// TIA Portal V16 program export: 1 tag tables, 0 data types, 20 data blocks, 10 code blocks (in call order from the OBs), 24 instance data blocks

VAR_GLOBAL   // PLC tag table "Default tag table"
   Iniciar_Manual AT %I0.0 : Bool;
   Detener_Manual AT %I0.1 : Bool;
   Raw_Temperatura AT %IW64 : Int;
   Raw_Humedad AT %IW66 : Int;
   Deshidratador AT %Q0.0 : Bool;
   Actuador AT %Q0.1 : Bool;
   Ventilador AT %Q0.2 : Bool;
   Resistencias AT %Q0.3 : Bool;
   Sensor_Modbus AT %Q0.4 : Bool;
   Sensor_HT AT %Q0.5 : Bool;
   System_Byte AT %MB1 : Byte;
   FirstScan AT %M1.0 : Bool;
   DiagStatusUpdate AT %M1.1 : Bool;
   AlwaysTRUE AT %M1.2 : Bool;
   AlwaysFALSE AT %M1.3 : Bool;
   Clock_Byte AT %MB0 : Byte;
   Clock_10Hz AT %M0.0 : Bool;
   Clock_5Hz AT %M0.1 : Bool;
   "Clock_2.5Hz" AT %M0.2 : Bool;
   Clock_2Hz AT %M0.3 : Bool;
   "Clock_1.25Hz" AT %M0.4 : Bool;
   Clock_1Hz AT %M0.5 : Bool;
   "Clock_0.625Hz" AT %M0.6 : Bool;
   "Clock_0.5Hz" AT %M0.7 : Bool;
   Control_Byte AT %MB2 : Byte;
   Detener AT %M2.0 : Bool;
   Iniciar AT %M2.1 : Bool;
   Pausar AT %M2.2 : Bool;
   Activar_Deshidratador AT %M2.3 : Bool;
   Limite_Matte AT %M2.6 : Bool;
   Sensor_Modbus_Manual AT %M2.4 : Bool;
   Set_Point_Deshidratador AT %MD4 : Real;
   Set_Point_Humedad AT %MD8 : Real;
   Iniciar_Pulse AT %M30.0 : Bool;
   Detener_Pulse AT %M30.1 : Bool;
   Guardar_Datos AT %M30.2 : Bool;
   Data_Log_Write_Error AT %M30.3 : Bool;
   Data_Log_Write_Busy AT %M30.4 : Bool;
   Data_Log_Write_Done AT %M30.5 : Bool;
   Data_Log_Write_Status AT %MW34 : Word;
   "Clock_0.016Hz" AT %M30.6 : Bool;
   Ret_Val AT %MW36 : Int;
   Sensor_HT_Manual AT %M2.5 : Bool;
   Actuador_Manual AT %M2.7 : Bool;
   Activar_Actuador AT %M3.0 : Bool;
   Tag_1 AT %M31.1 : Bool;
   Habilitar_Matte AT %M3.1 : Bool;
   Set_Point_Limite AT %MD12 : Real;
   Humedad_Material_D11 AT %MD38 : Real;
   Humedad_Material_D13 AT %MD42 : Real;
   Humedad_Material_D16 AT %MD46 : Real;
   Temp_D13 AT %MD54 : Real;
   Temp_Matte AT %MD58 : Real;
   Hum_Matte AT %MD62 : Real;
   Temp_D11 AT %MD50 : Real;
   Temp_Matte_Aux AT %MD66 : Real;
   Clock_Matte_Manual AT %M31.2 : Bool;
   Humedad_Material_D11_Ajuste AT %MD70 : Real;
   Humedad_Material_D13_Ajuste AT %MD74 : Real;
   Humedad_Material_D16_Ajuste AT %MD78 : Real;
   Hum_Matte_Aux AT %MD82 : Real;
   Random_Real_Seconds AT %MD86 : Real;
   Random_Status AT %MW90 : Int;
   Random_Sub_Status AT %MW92 : Int;
   Random_Error AT %M3.2 : Bool;
   Clock_Pulse AT %M3.3 : Bool;
   Randon_Dint_Seconds AT %MD94 : DInt;
   Tiempo_Histeresis_D1 AT %MD98 : Time;
   Set_Point_Deshidratador1_Inicial AT %MD102 : Real;
   Set_Point_Deshidratador1_Intermedia AT %MD106 : Real;
   Set_Point_Deshidratador1_Final AT %MD110 : Real;
   Set_Point_Humedad_D1_Inicial AT %MD114 : Real;
   Set_Point_Humedad_D1_Intermedia AT %MD118 : Real;
   Set_Point_Humedad_D1_Final AT %MD122 : Real;
   Detener_Desde_Modo_Preset AT %M31.3 : Bool;
END_VAR
VAR_GLOBAL CONSTANT   // user constants
   Set_Point_Temp_Default : Real := 55.0;
   Set_Pont_Hum_Default : Real := 5.0;
   Set_Point_Lim_Default : Real := -16.0;
   Aux_Hum_D1 : Real := 10.0;
   Aux_Hum_D4 : Real := 25.0;
   Aux_Hum_D8 : Real := 25.0;
END_VAR

DATA_BLOCK "Alarmas"   // DB44
{ S7_Optimized_Access := 'FALSE' }
VERSION : 0.1
   VAR
      Alarma_Fin_Operacion : Bool;
      Alarma_Fallo_Deh : Bool;
   END_VAR
BEGIN
END_DATA_BLOCK

DATA_BLOCK "CREAR_DB"   // DB7
{ S7_Optimized_Access := 'TRUE' }
VERSION : 0.1
   VAR
      records : UDInt := 17280;
      "name" : String := 'logging';
      id : DWord := 1;
      headers : String := 'HumD11,HumD13,HumD16,TempD11,TempD13,HumMatte,TempMatte';
      data : Struct
         humD11 : Real;
         humD13 : Real;
         humD16 : Real;
         tempD11 : Real;
         tempD13 : Real;
         humMatte : Real;
         tempMatte : Real;
      END_STRUCT;
      done : Bool;
      busy : Bool := true;
      error : Bool;
      status : Word;
   END_VAR
BEGIN
END_DATA_BLOCK

DATA_BLOCK "Calibracion_Sensores"   // DB31
{ S7_Optimized_Access := 'TRUE' }
VERSION : 0.1
   VAR
      Ajuste_D11 : Real := 1.0;
      Ajuste_D13 : Real := 1.0;
      Ajuste_D16 : Real := 1.0;
      Ajuste_T1 : Real := 1.0;
   END_VAR
BEGIN
END_DATA_BLOCK

DATA_BLOCK "Control_Log_DB"   // DB33
{ S7_Optimized_Access := 'FALSE' }
VERSION : 0.1
   VAR
      Iniciar_Log : Bool;
      Almacenar_Logs : Bool;
      Teminar_Log : Bool;
   END_VAR
BEGIN
END_DATA_BLOCK

DATA_BLOCK "DATOS_MODSEC"   // DB13
{ S7_Optimized_Access := 'TRUE' }
VERSION : 0.1
   VAR
      SimuHR : Int;
   END_VAR
   VAR RETAIN
      "Paso Control HR" : Time := T#5000ms;
      "Paso Grafica" : Time := T#10ms;
      "CRECIMIENTO HR" : Real := 80.0;
      TempMinHR : Real := 22.0;
   END_VAR
   VAR
      TempInf : Real := 0.0;
      TempSup : Real := 100.0;
      TempFilt : Real;
      TempFiltJP : Real;
      HRAux : Real;
      HRAuxJP : Real;
      HRFilt : Real;
      HRSim : Int;
      TempSim : Int;
      ProporcionHumedad : Real := 0.9;
      TempFiltCuar : Real;
      HRFiltCuar : Real;
      HRAuxCuar : Real;
   END_VAR
BEGIN
END_DATA_BLOCK

DATA_BLOCK "DATOS_VARIABLES"   // DB8
{ S7_Optimized_Access := 'FALSE' }
VERSION : 0.1
   VAR
      humD11 : Real;
      humD13 : Real;
      humD16 : Real;
      tempD11 : Real;
      tempD13 : Real;
      humMatte : Real;
      tempMatte : Real;
   END_VAR
BEGIN
END_DATA_BLOCK

DATA_BLOCK "MB_CONFIG"   // DB9
{ S7_Optimized_Access := 'FALSE' }
VERSION : 0.1
   VAR
      Again : Bool;
      Req : Bool;
      Mb_Addr : UInt := 1;
      Mode : USInt := 0;
      Data_Addr : UDInt := 40001;
      Data_Len : UInt := 5;
      Done : Bool;
      Busy : Bool;
      Error : Bool;
      Status : Word;
      Error_Status : Word;
      "Step" : Int := 1;
   END_VAR
BEGIN
END_DATA_BLOCK

DATA_BLOCK "MB_DATA_BUFFER"   // DB10
{ S7_Optimized_Access := 'FALSE' }
VERSION : 0.1
   VAR
      REGISTERS : Array[0..4] of UInt;
   END_VAR
BEGIN
END_DATA_BLOCK

DATA_BLOCK "MB_LOAD"   // DB11
{ S7_Optimized_Access := 'FALSE' }
VERSION : 0.1
   VAR
      Baud : UDInt := 9600;
      Parity : UDInt;
      Done : Bool;
      Error : Bool;
      Status : Word;
      Done_Stored : Bool;
      Error_Stored : Bool;
      Status_Error : Word;
   END_VAR
BEGIN
END_DATA_BLOCK

DATA_BLOCK "Modos_Operacion"   // DB32
{ S7_Optimized_Access := 'TRUE' }
VERSION : 0.1
   VAR
      Modo_Preset_D1 : Bool;
      Momento_Actual_D1 : Int;
   END_VAR
BEGIN
END_DATA_BLOCK

DATA_BLOCK "DB 333"   // DB333
{ S7_Optimized_Access := 'FALSE' }
AUTHOR : AWP_S7P
FAMILY : WEB
VERSION : 1.0
   VAR
      magic : DWord := DW#16#41575043;
      consistency_tag : DWord := DW#16#24B8E9AC;
      db_version : Word := W#16#0001;
      length : UInt := 4326;
      pagetab_of : UInt := 92;
      pagetab_count : UInt := 36;
      excludetab_of : UInt := 452;
      excludetab_count : UInt := 4;
      fragmentlist_of : UInt := 460;
      fragmentlist_count : UInt := 55;
      fragmenttab_of : UInt := 576;
      fragmenttab_count : UInt := 45;
      datatab_of : UInt := 1206;
      datatab_count : UInt := 30;
      usenametab_of : UInt := 1326;
      usenametab_count : UInt := 0;
      enumreftab_of : UInt := 1326;
      enumreftab_count : UInt := 0;
      enumtab_of : UInt := 1326;
      enumtab_count : UInt := 0;
      textlist_of : UInt := 1326;
      textlist_count : UInt := 3000;
      language_frag_tab_of : UInt := 570;
      language_frag_tab_count : UInt := 6;
      application_name : UInt := 1;
      application_url : UInt := 17;
      application_desc : UInt := 34;
      enum_defs_fragment_start : UInt := 0;
      enum_defs_fragment_count : UInt := 0;
      commandstate : Struct
         last_error : Int := 0;
         debug_mode : Int := 0;
         init : Bool := True;
         deactivate : Bool := False;
         initializing : Bool := False;
         error : Bool := False;
         deactivating : Bool := False;
         deactivated : Bool := False;
         initialized : Bool := False;
         reserved1 : Bool := False;
         reserved2 : Byte := B#16#00;
      END_STRUCT;
      requesttab : Array[1..4] of Struct
         page_index : UInt;
         fragment_index : UInt;
         continue : Bool;
         "repeat" : Bool;
         abort : Bool;
         finish : Bool;
         idle : Bool;
         waiting : Bool;
         sending : Bool;
         aborting : Bool;
         reserved3 : Byte;
      END_STRUCT;
      pagetab : Array[1..36] of Struct
         index : UInt;
         url : UInt;
         mime_type : UInt;
         fragment_start : UInt;
         fragment_num : UInt;
      END_STRUCT;
      excludetab : Array[1..4] of UInt;
      fragmentlist : Array[1..55] of UInt;
      language_frag_tab : Struct
         max_language : UInt := 0;
         fragment_count : UInt := 0;
         nolang_offset : UInt := 0;
      END_STRUCT;
      fragmenttab : Array[1..45] of Struct
         fragment_name : UInt;
         fragment_type : Byte;
         fragment_version : Byte;
         content_db : UInt;
         content_of : UInt;
         content_length : UInt;
         data_start : UInt;
         data_num : UInt;
      END_STRUCT;
      datatab : Array[1..30] of Struct
         variable_name : UInt;
         direction : Int;
      END_STRUCT;
      textlist : Array[1..3000] of Byte := 5365727669646F725175616E74756D0076696577735C6C6F67696E2E68746D6C005365727669646F725175616E74756D00494F4431487973745374617475732E68746D6C00746578742F68746D6C00494F44314D6F64652E68746D6C00746578742F68746D6C00494F44315374617475732E68746D6C00746578742F68746D6C00494F4465685374617475732E68746D6C00746578742F68746D6C00494F48756D4431312E68746D6C00746578742F68746D6C00494F48756D443146696E616C5374617475732E68746D6C00746578742F68746D6C00494F48756D4431496E69745374617475732E68746D6C00746578742F68746D6C00494F48756D44314D69645374617475732E68746D6C00746578742F68746D6C00494F48756D44315374617475732E68746D6C00746578742F68746D6C00494F53746172744465682E68746D6C00746578742F68746D6C00494F53746F704465682E68746D6C00746578742F68746D6C00494F54656D7044312E68746D6C00746578742F68746D6C00494F54656D70443146696E616C5374617475732E68746D6C00746578742F68746D6C00494F54656D704431496E69745374617475732E68746D6C00746578742F68746D6C00494F54656D7044314D69645374617475732E68746D6C00746578742F68746D6C00494F54656D7044315374617475732E68746D6C00746578742F68746D6C006E61764261722E68746D6C00746578742F68746D6C00736964654261722E68746D6C00746578742F68746D6C0076696577732F6373732F636F6E74726F6C2E63737300746578742F6373730076696577732F6373732F6C6F67696E2E63737300746578742F6373730076696577732F6373732F6E61765374796C652E63737300746578742F6373730076696577732F6373732F746F67676C655374796C652E63737300746578742F6373730076696577732F64617368626F6172644465682E68746D6C00746578742F68746D6C0076696577732F64617368626F61726448756D44312E68746D6C00746578742F68746D6C0076696577732F64617368626F61726454656D7044312E68746D6C00746578742F68746D6C0076696577732F64617461436F6E74726F6C2E68746D6C00746578742F68746D6C0076696577732F696D672F6C6F676F2E706E6700696D6167652F706E670076696577732F696E6465782E68746D6C00746578742F68746D6C0076696577732F6A732F64617368626F61726448756D44312E6A73006170706C69636174696F6E2F6A6176617363726970740076696577732F6A732F64617368626F61726454656D7044312E6A73006170706C69636174696F6E2F6A6176617363726970740076696577732F6A732F696E6465782E6A73006170706C69636174696F6E2F6A6176617363726970740076696577732F6A732F6A71756572792D332E332E312E6D696E2E6A73006170706C69636174696F6E2F6A6176617363726970740076696577732F6A732F6C6F67696E2E6A73006170706C69636174696F6E2F6A6176617363726970740076696577732F6A732F6E61765363726970742E6A73006170706C69636174696F6E2F6A6176617363726970740076696577732F6A732F736D6F6F74686965322E6A73006170706C69636174696F6E2F6A6176617363726970740076696577732F6C6F67696E2E68746D6C00746578742F68746D6C0076696577732F6373730076696577732F696D670076696577732F6A730076696577730076696577732F6373732F636F6E74726F6C2E6373730076696577732F6373732F6C6F67696E2E6373730076696577732F6373732F6E61765374796C652E6373730076696577732F6373732F746F67676C655374796C652E6373730076696577732F696D672F6C6F676F2E706E670076696577732F696D672F6C6F676F2E706E675F310076696577732F696D672F6C6F676F2E706E675F320076696577732F696D672F6C6F676F2E706E675F330076696577732F6A732F64617368626F61726448756D44312E6A730076696577732F6A732F64617368626F61726454656D7044312E6A730076696577732F6A732F696E6465782E6A730076696577732F6A732F6A71756572792D332E332E312E6D696E2E6A730076696577732F6A732F6A71756572792D332E332E312E6D696E2E6A735F310076696577732F6A732F6C6F67696E2E6A730076696577732F6A732F6E61765363726970742E6A730076696577732F6A732F736D6F6F74686965322E6A730076696577732F64617368626F6172644465682E68746D6C0076696577732F64617368626F6172644465682E68746D6C5F310076696577732F64617368626F61726448756D44312E68746D6C0076696577732F64617368626F61726448756D44312E68746D6C5F310076696577732F64617368626F61726454656D7044312E68746D6C0076696577732F64617368626F61726454656D7044312E68746D6C5F310076696577732F64617461436F6E74726F6C2E68746D6C0076696577732F64617461436F6E74726F6C2E68746D6C5F310076696577732F696E6465782E68746D6C0076696577732F696E6465782E68746D6C5F310076696577732F6C6F67696E2E68746D6C00494F4431487973745374617475732E68746D6C00494F44314D6F64652E68746D6C00494F44315374617475732E68746D6C00494F4465685374617475732E68746D6C00494F48756D4431312E68746D6C00494F48756D443146696E616C5374617475732E68746D6C00494F48756D4431496E69745374617475732E68746D6C00494F48756D44314D69645374617475732E68746D6C00494F48756D44315374617475732E68746D6C00494F53746172744465682E68746D6C00494F53746F704465682E68746D6C00494F54656D7044312E68746D6C00494F54656D70443146696E616C5374617475732E68746D6C00494F54656D704431496E69745374617475732E68746D6C00494F54656D7044314D69645374617475732E68746D6C00494F54656D7044315374617475732E68746D6C006E617642617200736964654261720022416374697661725F44657368696472617461646F722200225365745F506F696E745F44657368696472617461646F722200225365745F506F696E745F48756D6564616422002244657368696472617461646F72220022496E6963696172220022446574656E65722200224D6F646F735F4F7065726163696F6E222E4D6F646F5F5072657365745F443100225365745F506F696E745F44657368696472617461646F72315F496E696369616C2200225365745F506F696E745F44657368696472617461646F72315F496E7465726D656469612200225365745F506F696E745F44657368696472617461646F72315F46696E616C2200225365745F506F696E745F48756D656461645F44315F496E696369616C2200225365745F506F696E745F48756D656461645F44315F496E7465726D656469612200225365745F506F696E745F48756D656461645F44315F46696E616C2200225469656D706F5F486973746572657369735F44312200225469656D706F5F486973746572657369735F44312200224D6F646F735F4F7065726163696F6E222E4D6F646F5F5072657365745F44310022416374697661725F44657368696472617461646F7222002244657368696472617461646F722200224441544F535F5641524941424C4553222E68756D4D6174746500225365745F506F696E745F48756D656461645F44315F46696E616C2200225365745F506F696E745F48756D656461645F44315F496E696369616C2200225365745F506F696E745F48756D656461645F44315F496E7465726D656469612200225365745F506F696E745F48756D65646164220022496E6963696172220022446574656E65722200224441544F535F5641524941424C4553222E74656D704D6174746500225365745F506F696E745F44657368696472617461646F72315F46696E616C2200225365745F506F696E745F44657368696472617461646F72315F496E696369616C2200225365745F506F696E745F44657368696472617461646F72315F496E7465726D656469612200225365745F506F696E745F44657368696472617461646F72220000;
   END_VAR
BEGIN
   requesttab[1..4].page_index := 0;
   requesttab[1..4].fragment_index := 0;
   requesttab[1..4].continue := False;
   requesttab[1..4]."repeat" := False;
   requesttab[1..4].abort := False;
   requesttab[1..4].finish := False;
   requesttab[1..4].idle := False;
   requesttab[1..4].waiting := False;
   requesttab[1..4].sending := False;
   requesttab[1..4].aborting := False;
   requesttab[1..4].reserved3 := B#16#00;
   pagetab[1].index := 1;
   pagetab[2].index := 2;
   pagetab[3].index := 3;
   pagetab[4].index := 4;
   pagetab[5].index := 5;
   pagetab[6].index := 6;
   pagetab[7].index := 7;
   pagetab[8].index := 8;
   pagetab[9].index := 9;
   pagetab[10].index := 10;
   pagetab[11].index := 11;
   pagetab[12].index := 12;
   pagetab[13].index := 13;
   pagetab[14].index := 14;
   pagetab[15].index := 15;
   pagetab[16].index := 16;
   pagetab[17].index := 17;
   pagetab[18].index := 18;
   pagetab[19].index := 19;
   pagetab[20].index := 20;
   pagetab[21].index := 21;
   pagetab[22].index := 22;
   pagetab[23].index := 23;
   pagetab[24].index := 24;
   pagetab[25].index := 25;
   pagetab[26].index := 26;
   pagetab[27].index := 27;
   pagetab[28].index := 28;
   pagetab[29].index := 29;
   pagetab[30].index := 30;
   pagetab[31].index := 31;
   pagetab[32].index := 32;
   pagetab[33].index := 33;
   pagetab[34].index := 34;
   pagetab[35].index := 35;
   pagetab[36].index := 36;
   pagetab[1].url := 50;
   pagetab[2].url := 80;
   pagetab[3].url := 104;
   pagetab[4].url := 130;
   pagetab[5].url := 157;
   pagetab[6].url := 181;
   pagetab[7].url := 215;
   pagetab[8].url := 248;
   pagetab[9].url := 280;
   pagetab[10].url := 309;
   pagetab[11].url := 335;
   pagetab[12].url := 360;
   pagetab[13].url := 384;
   pagetab[14].url := 419;
   pagetab[15].url := 453;
   pagetab[16].url := 486;
   pagetab[17].url := 516;
   pagetab[18].url := 538;
   pagetab[19].url := 561;
   pagetab[20].url := 592;
   pagetab[21].url := 621;
   pagetab[22].url := 653;
   pagetab[23].url := 688;
   pagetab[24].url := 722;
   pagetab[25].url := 758;
   pagetab[26].url := 795;
   pagetab[27].url := 828;
   pagetab[28].url := 857;
   pagetab[29].url := 884;
   pagetab[30].url := 934;
   pagetab[31].url := 985;
   pagetab[32].url := 1026;
   pagetab[33].url := 1078;
   pagetab[34].url := 1119;
   pagetab[35].url := 1164;
   pagetab[36].url := 1209;
   pagetab[1].mime_type := 70;
   pagetab[2].mime_type := 94;
   pagetab[3].mime_type := 120;
   pagetab[4].mime_type := 147;
   pagetab[5].mime_type := 171;
   pagetab[6].mime_type := 205;
   pagetab[7].mime_type := 238;
   pagetab[8].mime_type := 270;
   pagetab[9].mime_type := 299;
   pagetab[10].mime_type := 325;
   pagetab[11].mime_type := 350;
   pagetab[12].mime_type := 374;
   pagetab[13].mime_type := 409;
   pagetab[14].mime_type := 443;
   pagetab[15].mime_type := 476;
   pagetab[16].mime_type := 506;
   pagetab[17].mime_type := 528;
   pagetab[18].mime_type := 551;
   pagetab[19].mime_type := 583;
   pagetab[20].mime_type := 612;
   pagetab[21].mime_type := 644;
   pagetab[22].mime_type := 679;
   pagetab[23].mime_type := 712;
   pagetab[24].mime_type := 748;
   pagetab[25].mime_type := 785;
   pagetab[26].mime_type := 818;
   pagetab[27].mime_type := 847;
   pagetab[28].mime_type := 874;
   pagetab[29].mime_type := 911;
   pagetab[30].mime_type := 962;
   pagetab[31].mime_type := 1003;
   pagetab[32].mime_type := 1055;
   pagetab[33].mime_type := 1096;
   pagetab[34].mime_type := 1141;
   pagetab[35].mime_type := 1186;
   pagetab[36].mime_type := 1226;
   pagetab[1].fragment_start := 1;
   pagetab[2].fragment_start := 2;
   pagetab[3].fragment_start := 3;
   pagetab[4].fragment_start := 4;
   pagetab[5].fragment_start := 5;
   pagetab[6].fragment_start := 6;
   pagetab[7].fragment_start := 7;
   pagetab[8].fragment_start := 8;
   pagetab[9].fragment_start := 9;
   pagetab[10].fragment_start := 10;
   pagetab[11].fragment_start := 11;
   pagetab[12].fragment_start := 12;
   pagetab[13].fragment_start := 13;
   pagetab[14].fragment_start := 14;
   pagetab[15].fragment_start := 15;
   pagetab[16].fragment_start := 16;
   pagetab[17].fragment_start := 17;
   pagetab[18].fragment_start := 18;
   pagetab[19].fragment_start := 19;
   pagetab[20].fragment_start := 20;
   pagetab[21].fragment_start := 21;
   pagetab[22].fragment_start := 22;
   pagetab[23].fragment_start := 23;
   pagetab[24].fragment_start := 27;
   pagetab[25].fragment_start := 31;
   pagetab[26].fragment_start := 35;
   pagetab[27].fragment_start := 39;
   pagetab[28].fragment_start := 43;
   pagetab[29].fragment_start := 47;
   pagetab[30].fragment_start := 48;
   pagetab[31].fragment_start := 49;
   pagetab[32].fragment_start := 50;
   pagetab[33].fragment_start := 52;
   pagetab[34].fragment_start := 53;
   pagetab[35].fragment_start := 54;
   pagetab[36].fragment_start := 55;
   pagetab[1..22].fragment_num := 1;
   pagetab[23..28].fragment_num := 4;
   pagetab[29..31].fragment_num := 1;
   pagetab[32].fragment_num := 2;
   pagetab[33..36].fragment_num := 1;
   excludetab[1] := 1236;
   excludetab[2] := 1246;
   excludetab[3] := 1256;
   excludetab[4] := 1265;
   fragmentlist[1] := 28;
   fragmentlist[2] := 29;
   fragmentlist[3] := 30;
   fragmentlist[4] := 31;
   fragmentlist[5] := 32;
   fragmentlist[6] := 33;
   fragmentlist[7] := 34;
   fragmentlist[8] := 35;
   fragmentlist[9] := 36;
   fragmentlist[10] := 37;
   fragmentlist[11] := 38;
   fragmentlist[12] := 39;
   fragmentlist[13] := 40;
   fragmentlist[14] := 41;
   fragmentlist[15] := 42;
   fragmentlist[16] := 43;
   fragmentlist[17] := 44;
   fragmentlist[18] := 45;
   fragmentlist[19] := 1;
   fragmentlist[20] := 2;
   fragmentlist[21] := 3;
   fragmentlist[22] := 4;
   fragmentlist[23] := 17;
   fragmentlist[24] := 44;
   fragmentlist[25] := 45;
   fragmentlist[26] := 18;
   fragmentlist[27] := 19;
   fragmentlist[28] := 44;
   fragmentlist[29] := 45;
   fragmentlist[30] := 20;
   fragmentlist[31] := 21;
   fragmentlist[32] := 44;
   fragmentlist[33] := 45;
   fragmentlist[34] := 22;
   fragmentlist[35] := 23;
   fragmentlist[36] := 44;
   fragmentlist[37] := 45;
   fragmentlist[38] := 24;
   fragmentlist[39] := 5;
   fragmentlist[40] := 6;
   fragmentlist[41] := 7;
   fragmentlist[42] := 8;
   fragmentlist[43] := 25;
   fragmentlist[44] := 44;
   fragmentlist[45] := 45;
   fragmentlist[46] := 26;
   fragmentlist[47] := 9;
   fragmentlist[48] := 10;
   fragmentlist[49] := 11;
   fragmentlist[50] := 12;
   fragmentlist[51] := 13;
   fragmentlist[52] := 14;
   fragmentlist[53] := 15;
   fragmentlist[54] := 16;
   fragmentlist[55] := 27;
   fragmenttab[1].fragment_name := 1271;
   fragmenttab[2].fragment_name := 1293;
   fragmenttab[3].fragment_name := 1313;
   fragmenttab[4].fragment_name := 1336;
   fragmenttab[5].fragment_name := 1362;
   fragmenttab[6].fragment_name := 1381;
   fragmenttab[7].fragment_name := 1402;
   fragmenttab[8].fragment_name := 1423;
   fragmenttab[9].fragment_name := 1444;
   fragmenttab[10].fragment_name := 1471;
   fragmenttab[11].fragment_name := 1499;
   fragmenttab[12].fragment_name := 1517;
   fragmenttab[13].fragment_name := 1546;
   fragmenttab[14].fragment_name := 1577;
   fragmenttab[15].fragment_name := 1595;
   fragmenttab[16].fragment_name := 1617;
   fragmenttab[17].fragment_name := 1639;
   fragmenttab[18].fragment_name := 1663;
   fragmenttab[19].fragment_name := 1689;
   fragmenttab[20].fragment_name := 1715;
   fragmenttab[21].fragment_name := 1743;
   fragmenttab[22].fragment_name := 1770;
   fragmenttab[23].fragment_name := 1799;
   fragmenttab[24].fragment_name := 1822;
   fragmenttab[25].fragment_name := 1847;
   fragmenttab[26].fragment_name := 1864;
   fragmenttab[27].fragment_name := 1883;
   fragmenttab[28].fragment_name := 1900;
   fragmenttab[29].fragment_name := 1920;
   fragmenttab[30].fragment_name := 1934;
   fragmenttab[31].fragment_name := 1950;
   fragmenttab[32].fragment_name := 1967;
   fragmenttab[33].fragment_name := 1981;
   fragmenttab[34].fragment_name := 2005;
   fragmenttab[35].fragment_name := 2028;
   fragmenttab[36].fragment_name := 2050;
   fragmenttab[37].fragment_name := 2069;
   fragmenttab[38].fragment_name := 2085;
   fragmenttab[39].fragment_name := 2100;
   fragmenttab[40].fragment_name := 2114;
   fragmenttab[41].fragment_name := 2139;
   fragmenttab[42].fragment_name := 2163;
   fragmenttab[43].fragment_name := 2186;
   fragmenttab[44].fragment_name := 2206;
   fragmenttab[45].fragment_name := 2213;
   fragmenttab[1..45].fragment_type := B#16#00;
   fragmenttab[1..45].fragment_version := B#16#00;
   fragmenttab[1..4].content_db := 334;
   fragmenttab[5].content_db := 335;
   fragmenttab[6].content_db := 336;
   fragmenttab[7].content_db := 337;
   fragmenttab[8..11].content_db := 338;
   fragmenttab[12].content_db := 339;
   fragmenttab[13..15].content_db := 340;
   fragmenttab[16..25].content_db := 341;
   fragmenttab[26..43].content_db := 342;
   fragmenttab[44..45].content_db := 334;
   fragmenttab[1].content_of := 1622;
   fragmenttab[2].content_of := 2684;
   fragmenttab[3].content_of := 3088;
   fragmenttab[4].content_of := 7122;
   fragmenttab[5..8].content_of := 8;
   fragmenttab[9].content_of := 10854;
   fragmenttab[10].content_of := 13240;
   fragmenttab[11].content_of := 14804;
   fragmenttab[12..13].content_of := 8;
   fragmenttab[14].content_of := 21410;
   fragmenttab[15].content_of := 22558;
   fragmenttab[16].content_of := 8;
   fragmenttab[17].content_of := 46036;
   fragmenttab[18].content_of := 48330;
   fragmenttab[19].content_of := 49986;
   fragmenttab[20].content_of := 51444;
   fragmenttab[21].content_of := 52014;
   fragmenttab[22].content_of := 53474;
   fragmenttab[23].content_of := 54046;
   fragmenttab[24].content_of := 58890;
   fragmenttab[25].content_of := 62442;
   fragmenttab[26].content_of := 8;
   fragmenttab[27].content_of := 6822;
   fragmenttab[28].content_of := 10574;
   fragmenttab[29].content_of := 10756;
   fragmenttab[30].content_of := 10942;
   fragmenttab[31].content_of := 11120;
   fragmenttab[32].content_of := 11292;
   fragmenttab[33].content_of := 11472;
   fragmenttab[34].content_of := 11664;
   fragmenttab[35].content_of := 11856;
   fragmenttab[36].content_of := 12050;
   fragmenttab[37].content_of := 12228;
   fragmenttab[38].content_of := 12392;
   fragmenttab[39].content_of := 12556;
   fragmenttab[40].content_of := 12736;
   fragmenttab[41].content_of := 12932;
   fragmenttab[42].content_of := 13130;
   fragmenttab[43].content_of := 13330;
   fragmenttab[44].content_of := 8;
   fragmenttab[45].content_of := 384;
   fragmenttab[1].content_length := 1061;
   fragmenttab[2].content_length := 403;
   fragmenttab[3].content_length := 4034;
   fragmenttab[4].content_length := 1146;
   fragmenttab[5..7].content_length := 65526;
   fragmenttab[8].content_length := 10845;
   fragmenttab[9].content_length := 2386;
   fragmenttab[10].content_length := 1564;
   fragmenttab[11].content_length := 6294;
   fragmenttab[12].content_length := 65526;
   fragmenttab[13].content_length := 21401;
   fragmenttab[14].content_length := 1148;
   fragmenttab[15].content_length := 149;
   fragmenttab[16].content_length := 46027;
   fragmenttab[17].content_length := 2294;
   fragmenttab[18].content_length := 1656;
   fragmenttab[19].content_length := 1457;
   fragmenttab[20].content_length := 570;
   fragmenttab[21].content_length := 1460;
   fragmenttab[22].content_length := 571;
   fragmenttab[23].content_length := 4843;
   fragmenttab[24].content_length := 3552;
   fragmenttab[25].content_length := 1448;
   fragmenttab[26].content_length := 6814;
   fragmenttab[27].content_length := 3752;
   fragmenttab[28].content_length := 181;
   fragmenttab[29].content_length := 185;
   fragmenttab[30].content_length := 178;
   fragmenttab[31].content_length := 171;
   fragmenttab[32].content_length := 179;
   fragmenttab[33].content_length := 191;
   fragmenttab[34].content_length := 192;
   fragmenttab[35].content_length := 194;
   fragmenttab[36].content_length := 177;
   fragmenttab[37].content_length := 164;
   fragmenttab[38].content_length := 163;
   fragmenttab[39].content_length := 180;
   fragmenttab[40].content_length := 196;
   fragmenttab[41].content_length := 197;
   fragmenttab[42].content_length := 199;
   fragmenttab[43].content_length := 184;
   fragmenttab[44].content_length := 375;
   fragmenttab[45].content_length := 1237;
   fragmenttab[1..24].data_start := 0;
   fragmenttab[25].data_start := 1;
   fragmenttab[26..27].data_start := 0;
   fragmenttab[28].data_start := 15;
   fragmenttab[29].data_start := 16;
   fragmenttab[30].data_start := 17;
   fragmenttab[31].data_start := 18;
   fragmenttab[32].data_start := 19;
   fragmenttab[33].data_start := 20;
   fragmenttab[34].data_start := 21;
   fragmenttab[35].data_start := 22;
   fragmenttab[36].data_start := 23;
   fragmenttab[37].data_start := 24;
   fragmenttab[38].data_start := 25;
   fragmenttab[39].data_start := 26;
   fragmenttab[40].data_start := 27;
   fragmenttab[41].data_start := 28;
   fragmenttab[42].data_start := 29;
   fragmenttab[43].data_start := 30;
   fragmenttab[44..45].data_start := 0;
   fragmenttab[1..24].data_num := 0;
   fragmenttab[25].data_num := 14;
   fragmenttab[26..27].data_num := 0;
   fragmenttab[28..43].data_num := 1;
   fragmenttab[44..45].data_num := 0;
   datatab[1].variable_name := 2221;
   datatab[2].variable_name := 2245;
   datatab[3].variable_name := 2271;
   datatab[4].variable_name := 2291;
   datatab[5].variable_name := 2307;
   datatab[6].variable_name := 2317;
   datatab[7].variable_name := 2327;
   datatab[8].variable_name := 2360;
   datatab[9].variable_name := 2395;
   datatab[10].variable_name := 2433;
   datatab[11].variable_name := 2466;
   datatab[12].variable_name := 2497;
   datatab[13].variable_name := 2531;
   datatab[14].variable_name := 2560;
   datatab[15].variable_name := 2583;
   datatab[16].variable_name := 2606;
   datatab[17].variable_name := 2639;
   datatab[18].variable_name := 2663;
   datatab[19].variable_name := 2679;
   datatab[20].variable_name := 2706;
   datatab[21].variable_name := 2735;
   datatab[22].variable_name := 2766;
   datatab[23].variable_name := 2800;
   datatab[24].variable_name := 2820;
   datatab[25].variable_name := 2830;
   datatab[26].variable_name := 2840;
   datatab[27].variable_name := 2868;
   datatab[28].variable_name := 2901;
   datatab[29].variable_name := 2936;
   datatab[30].variable_name := 2974;
   datatab[1..14].direction := 2;
   datatab[15..30].direction := 3;
END_DATA_BLOCK

DATA_BLOCK "DB 334"   // DB334
{ S7_Optimized_Access := 'FALSE' }
AUTHOR : AWP_S7P
FAMILY : WEB
VERSION : 0.1
   VAR
      MAGIC : DWord := DW#16#4157_5046;
      CONSISTENCY_TAG : DWord := 616098220;
      TEMP_1 : Array[1..375] of Byte := 0A3C6E617620636C6173733D226E6176626172206E61766261722D637573746F6D223E0A093C64697620636C6173733D22636F6E7461696E65722D666C756964223E0A09093C64697620636C6173733D226E61766261722D686561646572223E0A0909093C6120636C6173733D226E61766261722D6272616E642220687265663D222F6177702F5365727669646F725175616E74756D2F76696577732F696E6465782E68746D6C223E0A090909093C696D672069643D226C6F676F2D696D6722207372633D22696D672F6C6F676F2E706E67223E0A0909093C2F613E0A0909093C627574746F6E20747970653D22627574746F6E2220636C6173733D2262746E2062746E2D64616E676572206E61766261722D62746E206E61766261722D7269676874223E3C6120687265663D222F466F726D4C6F67696E3F4C4F474F5554223E53414C49523C2F613E3C2F627574746F6E3E2020202020202020202020200A09093C2F6469763E0A093C2F6469763E0A3C2F6E61763E;
      TEMP_2 : Array[1..1237] of Byte := 0A3C6469762069643D2277726170706572223E0A093C64697620636C6173733D226F7665726C6179223E3C2F6469763E0A0A093C6E617620636C6173733D226E6176626172206E61766261722D696E7665727365206E61766261722D66697865642D746F70222069643D22736964656261722D777261707065722220726F6C653D226E617669676174696F6E223E0A09093C756C20636C6173733D226E617620736964656261722D6E6176223E0A0909093C6C6920636C6173733D22736964656261722D6272616E64223E0A090909093C6120687265663D222F6177702F5365727669646F725175616E74756D2F76696577732F636F6E74726F6C4465682E68746D6C223E0A090909092020203C696D672069643D226C6F676F2D696D6722207372633D22696D672F6C6F676F2E706E67222077696474683D2231353022206865696768743D223730223E0A090909093C2F613E0A0909093C2F6C693E0A0909093C6C6920636C6173733D2264726F70646F776E2D6D61696E223E0A09090920203C6120687265663D22232220636C6173733D2264726F70646F776E2D746F67676C652220646174612D746F67676C653D2264726F70646F776E223E446573686964726174616369C3B36E203C7370616E20636C6173733D226361726574223E3C2F7370616E3E3C2F613E0A09090920203C756C20636C6173733D2264726F70646F776E2D6D656E752220726F6C653D226D656E75223E0A090909093C6C693E3C6120687265663D222F6177702F5365727669646F725175616E74756D2F76696577732F636F6E74726F6C4465682E68746D6C223E436F6E74726F6C2044657368696472617461646F7265733C2F613E3C2F6C693E0A090909093C6C693E3C6120687265663D222F6177702F5365727669646F725175616E74756D2F76696577732F64617368626F6172644465682E68746D6C223E436F6E74726F6C20416D6269656E74653C2F613E3C2F6C693E0A09090920203C2F756C3E0A0909093C2F6C693E0A0909093C6C6920636C6173733D2264726F70646F776E2D6D61696E223E0A09090920203C6120687265663D22232220636C6173733D2264726F70646F776E2D746F67676C652220646174612D746F67676C653D2264726F70646F776E223E426C6F636B636861696E203C7370616E20636C6173733D226361726574223E3C2F7370616E3E3C2F613E0A09090920203C756C20636C6173733D2264726F70646F776E2D6D656E752220726F6C653D226D656E75223E0A090909093C6C693E3C6120687265663D222F6177702F5365727669646F725175616E74756D2F76696577732F64617461436F6E74726F6C2E68746D6C223E436F6E74726F6C204461746F733C2F613E3C2F6C693E0A09090920203C2F756C3E0A0909093C2F6C693E202020202020202020202020202020200A09093C2F756C3E0A093C2F6E61763E0A0A093C6469762069643D22706167652D636F6E74656E742D77726170706572223E0A09093C627574746F6E20747970653D22627574746F6E2220636C6173733D2262746E2062746E2D6C6720637573746F6D2D62746E2220646174612D746F67676C653D226F666663616E766173223E0A090909416363696F6E657320203C6920636C6173733D2266612066612D62617273223E3C2F693E0A09093C2F627574746F6E3E0A093C2F6469763E0A0A3C2F6469763E;
      TEMP_3 : Array[1..1061] of Byte := 68746D6C2C0D0A2E636F6C666F726D207B20666C6F61743A6C6566743B2077696474683A3530253B7D0D0A0D0A3A726F6F74207B0D0A202020202D2D636F6C6F722D677265656E3A20233030613837383B0D0A202020202D2D636F6C6F722D7265643A20236665356534313B0D0A202020202D2D636F6C6F722D627574746F6E3A20236664666666663B0D0A202020202D2D636F6C6F722D626C61636B3A20233030303B0D0A7D0D0A2E7377697463682D627574746F6E207B0D0A20202020646973706C61793A20696E6C696E652D626C6F636B3B0D0A7D0D0A2E7377697463682D627574746F6E202E7377697463682D627574746F6E5F5F636865636B626F78207B0D0A20202020646973706C61793A206E6F6E653B0D0A7D0D0A2E7377697463682D627574746F6E202E7377697463682D627574746F6E5F5F6C6162656C207B0D0A202020206261636B67726F756E642D636F6C6F723A20766172282D2D636F6C6F722D726564293B0D0A2020202077696474683A203472656D3B0D0A202020206865696768743A203272656D3B0D0A20202020626F726465722D7261646975733A203272656D3B0D0A20202020646973706C61793A20696E6C696E652D626C6F636B3B0D0A20202020706F736974696F6E3A2072656C61746976653B0D0A7D0D0A2E7377697463682D627574746F6E202E7377697463682D627574746F6E5F5F6C6162656C3A6265666F7265207B0D0A202020207472616E736974696F6E3A202E32733B0D0A20202020646973706C61793A20626C6F636B3B0D0A20202020706F736974696F6E3A206162736F6C7574653B0D0A2020202077696474683A203272656D3B0D0A202020206865696768743A203272656D3B0D0A202020206261636B67726F756E642D636F6C6F723A20766172282D2D636F6C6F722D627574746F6E293B0D0A20202020636F6E74656E743A2027273B0D0A20202020626F726465722D7261646975733A203530253B0D0A20202020626F782D736861646F773A20696E7365742030707820307078203070782031707820766172282D2D636F6C6F722D626C61636B293B0D0A7D0D0A2E7377697463682D627574746F6E202E7377697463682D627574746F6E5F5F636865636B626F783A636865636B6564202B202E7377697463682D627574746F6E5F5F6C6162656C207B0D0A202020206261636B67726F756E642D636F6C6F723A20766172282D2D636F6C6F722D677265656E293B0D0A7D0D0A2E7377697463682D627574746F6E202E7377697463682D627574746F6E5F5F636865636B626F783A636865636B6564202B202E7377697463682D627574746F6E5F5F6C6162656C3A6265666F7265207B0D0A202020207472616E73666F726D3A207472616E736C61746558283272656D293B0D0A7D0D0A2E636F6E7461696E65724872207B0D0A2009646973706C61793A20666C65783B200D0A7D;
      TEMP_4 : Array[1..403] of Byte := 68746D6C2C0D0A626F6479207B0D0A20206865696768743A20313030253B0D0A7D0D0A0D0A626F6479207B0D0A2020646973706C61793A202D6D732D666C6578626F783B0D0A2020646973706C61793A202D7765626B69742D626F783B0D0A2020646973706C61793A20666C65783B0D0A20202D6D732D666C65782D616C69676E3A2063656E7465723B0D0A20202D6D732D666C65782D7061636B3A2063656E7465723B0D0A20202D7765626B69742D626F782D616C69676E3A2063656E7465723B0D0A2020616C69676E2D6974656D733A2063656E7465723B0D0A20202D7765626B69742D626F782D7061636B3A2063656E7465723B0D0A20206A7573746966792D636F6E74656E743A2063656E7465723B0D0A202070616464696E672D746F703A20343070783B0D0A202070616464696E672D626F74746F6D3A20343070783B0D0A20206261636B67726F756E642D696D6167653A206C696E6561722D6772616469656E7428726762283235352C203235352C20323535292C7267622836302C2036312C20353929293B0D0A7D0D0A2020;
      TEMP_5 : Array[1..4034] of Byte := 2F2A2043535320446F63756D656E74202A2F0D0A0D0A626F6479207B0D0A20202020706F736974696F6E3A2072656C61746976653B0D0A202020206F766572666C6F772D783A2068696464656E3B0D0A7D0D0A0D0A626F64792C0D0A68746D6C207B206865696768743A20313030253B7D0D0A2E6E6176202E6F70656E203E20612C200D0A2E6E6176202E6F70656E203E20613A686F7665722C200D0A2E6E6176202E6F70656E203E20613A666F637573207B6261636B67726F756E642D636F6C6F723A207472616E73706172656E743B7D0D0A0D0A2377726170706572207B0D0A2020202070616464696E672D6C6566743A20303B0D0A202020202D7765626B69742D7472616E736974696F6E3A20616C6C20302E357320656173653B0D0A202020202D6D6F7A2D7472616E736974696F6E3A20616C6C20302E357320656173653B0D0A202020202D6F2D7472616E736974696F6E3A20616C6C20302E357320656173653B0D0A202020207472616E736974696F6E3A20616C6C20302E357320656173653B0D0A7D0D0A0D0A23777261707065722E746F67676C65647B0D0A0970616464696E672D6C6566743A2032323070783B0D0A7D0D0A0D0A23736964656261722D77726170706572207B0D0A202020207A2D696E6465783A20313030303B0D0A202020206C6566743A2032323070783B0D0A2020202077696474683A20303B0D0A202020206865696768743A20313030253B0D0A202020206D617267696E2D6C6566743A202D32323070783B0D0A202020206F766572666C6F772D793A206175746F3B0D0A202020206F766572666C6F772D783A2068696464656E3B0D0A202020206261636B67726F756E643A206C696E6561722D6772616469656E74287267622836302C2036312C203539292C726762283235342C203235352C2032353529293B0D0A202020202D7765626B69742D7472616E736974696F6E3A20616C6C20302E357320656173653B0D0A202020202D6D6F7A2D7472616E736974696F6E3A20616C6C20302E357320656173653B0D0A202020202D6F2D7472616E736974696F6E3A20616C6C20302E357320656173653B0D0A202020207472616E736974696F6E3A20616C6C20302E357320656173653B0D0A7D0D0A0D0A23736964656261722D777261707065723A3A2D7765626B69742D7363726F6C6C626172207B0D0A20202020646973706C61793A206E6F6E653B0D0A7D0D0A0D0A23777261707065722E746F67676C65642023736964656261722D77726170706572207B0D0A2020202077696474683A2032323070783B0D0A7D0D0A0D0A23706167652D636F6E74656E742D77726170706572207B0D0A2020202077696474683A20313030253B0D0A2020202070616464696E672D746F703A20313570783B0D0A2020202070616464696E672D626F74746F6D3A20313070783B0D0A7D0D0A0D0A23777261707065722E746F67676C65642023706167652D636F6E74656E742D77726170706572207B0D0A20202020706F736974696F6E3A206162736F6C7574653B0D0A202020206D617267696E2D72696768743A202D32323070783B0D0A7D0D0A0D0A236C6F676F75745F736964656261725F627574746F6E207B0D0A20202020706F736974696F6E3A206162736F6C7574653B0D0A20202020646973706C61793A20696E6C696E652D626C6F636B3B0D0A2020202077696474683A2032323070783B0D0A20202020626F74746F6D3A20303B0D0A7D0D0A0D0A2E6E61766261722D637573746F6D207B0D0A202020206865696768743A2032303070783B0D0A202020206261636B67726F756E643A206C696E6561722D6772616469656E7428746F2072696768742C207267622836302C2036312C203539292C726762283235342C203235352C2032353529293B0D0A20202020636F6C6F723A3333333B0D0A20202020626F726465722D7261646975733A303B0D0A7D0D0A0D0A2E736964656261722D6E6176207B0D0A20202020706F736974696F6E3A206162736F6C7574653B0D0A20202020746F703A20303B0D0A2020202077696474683A2032323070783B0D0A202020206D617267696E3A20303B0D0A2020202070616464696E673A20303B0D0A202020206C6973742D7374796C653A206E6F6E653B0D0A7D0D0A0D0A2E736964656261722D6E6176206C69207B0D0A20202020706F736974696F6E3A2072656C61746976653B200D0A202020206C696E652D6865696768743A20323070783B0D0A20202020646973706C61793A20696E6C696E652D626C6F636B3B0D0A2020202077696474683A20313030253B0D0A202020206D617267696E2D6C6566743A20313070783B2020202020200D0A7D0D0A0D0A2E736964656261722D6E61762D6D61696E206C69207B0D0A20202020706F736974696F6E3A2072656C61746976653B200D0A202020206C696E652D6865696768743A20323070783B0D0A20202020646973706C61793A20696E6C696E652D626C6F636B3B0D0A2020202077696474683A20313030253B2020202020200D0A7D0D0A0D0A2E736964656261722D6E6176206C693A6265666F7265207B0D0A20202020636F6E74656E743A2027273B0D0A20202020706F736974696F6E3A206162736F6C7574653B0D0A20202020746F703A20303B0D0A202020206C6566743A20303B0D0A202020207A2D696E6465783A202D313B0D0A202020206865696768743A20313030253B0D0A2020202077696474683A203370783B0D0A202020206261636B67726F756E642D636F6C6F723A20233343334433443B0D0A202020202D7765626B69742D7472616E736974696F6E3A207769647468202E327320656173652D696E3B0D0A2020202020202D6D6F7A2D7472616E736974696F6E3A20207769647468202E327320656173652D696E3B0D0A202020202020202D6D732D7472616E736974696F6E3A20207769647468202E327320656173652D696E3B0D0A2020202020202020202020207472616E736974696F6E3A207769647468202E327320656173652D696E3B0D0A7D0D0A0D0A2E736964656261722D6E6176206C693A686F7665723A6265666F72652C0D0A2E736964656261722D6E6176206C692E6F70656E3A686F7665723A6265666F72657B0D0A0977696474683A20313030253B0D0A092D7765626B69742D7472616E736974696F6E3A207769647468202E327320656173652D696E3B0D0A2020202020202D6D6F7A2D7472616E736974696F6E3A20207769647468202E327320656173652D696E3B0D0A202020202020202D6D732D7472616E736974696F6E3A20207769647468202E327320656173652D696E3B0D0A2020202020202020202020207472616E736974696F6E3A207769647468202E327320656173652D696E3B0D0A7D0D0A0D0A2E736964656261722D6E6176206C6920617B0D0A09646973706C61793A20626C6F636B3B0D0A09636F6C6F723A20234646463B0D0A09746578742D6465636F726174696F6E3A206E6F6E653B0D0A0970616464696E673A20313070782031357078203130707820333070783B0D0A7D0D0A0D0A2E736964656261722D6E6176206C6920613A686F7665722C0D0A2E736964656261722D6E6176206C6920613A6163746976652C0D0A2E736964656261722D6E6176206C6920613A666F6375732C0D0A2E736964656261722D6E6176206C692E6F70656E20613A686F7665722C0D0A2E736964656261722D6E6176206C692E6F70656E20613A6163746976652C0D0A2E736964656261722D6E6176206C692E6F70656E20613A666F6375737B0D0A09636F6C6F723A20234646463B0D0A09746578742D6465636F726174696F6E3A206E6F6E653B0D0A096261636B67726F756E642D636F6C6F723A207472616E73706172656E743B0D0A7D0D0A0D0A2E736964656261722D6E6176203E202E736964656261722D6272616E647B0D0A096865696768743A20393070783B0D0A09666F6E742D73697A653A20323270783B0D0A096C696E652D6865696768743A20343670783B0D0A202020206D617267696E2D6C6566743A203070783B200D0A7D0D0A0D0A2E736964656261722D6E6176203E202E64726F70646F776E2D6D61696E7B0D0A202020206D617267696E2D6C6566743A203070783B200D0A7D0D0A0D0A2E736964656261722D6E6176202E64726F70646F776E2D6D656E757B0D0A09706F736974696F6E3A2072656C61746976653B0D0A0977696474683A20313030253B0D0A0970616464696E673A20303B0D0A096D617267696E3A20303B0D0A09626F726465722D7261646975733A20303B0D0A09626F726465723A6E6F6E653B0D0A096261636B67726F756E643A206C696E6561722D6772616469656E74287267622836302C2036312C203539292C726762283235352C203235352C2032353529293B0D0A09626F782D736861646F773A206E6F6E653B0D0A7D0D0A0D0A2E637573746F6D2D62746E7B0D0A096D617267696E2D6C6566743A20313570783B0D0A09636F6C6F723A20233343334433443B0D0A096261636B67726F756E642D636F6C6F723A20234646464646463B0D0A7D0D0A0D0A2E637573746F6D2D62746E3A686F7665727B0D0A096D617267696E2D6C6566743A20313570783B0D0A09636F6C6F723A2077686974653B0D0A096261636B67726F756E642D636F6C6F723A20233343334433443B0D0A7D0D0A0D0A2E636F6E7461696E65724872207B0D0A20202020646973706C61793A20666C65783B0D0A20202020666C65782D646972656374696F6E3A20726F773B200D0A7D0D0A0D0A2E6E61766261722D6C69676874202E6E61766261722D6272616E64207B0D0A20202020636F6C6F723A20233343334433443B0D0A7D0D0A0D0A2E6E61766261722D637573746F6D202E6E61766261722D6272616E64207B0D0A20202070616464696E673A20337078203770783B0D0A202020636F6C6F723A20233343334433443B0D0A2020206865696768743A2032303070783B0D0A7D0D0A0D0A2E6E61766261722D637573746F6D20627574746F6E20617B0D0A20202020636F6C6F723A20233343334433443B0D0A7D0D0A0D0A2E6E61766261722D636F6C6C617073652E636F6C6C61707365207B0D0A20202020646973706C61793A20626C6F636B21696D706F7274616E743B0D0A7D0D0A0D0A2E6E61766261722D6E61763E6C692C202E6E61766261722D6E6176207B0D0A20202020666C6F61743A206C6566742021696D706F7274616E743B0D0A7D0D0A0D0A2E6E61766261722D6E61762E6E61766261722D72696768743A6C6173742D6368696C64207B0D0A202020206D617267696E2D72696768743A202D313570782021696D706F7274616E743B0D0A7D0D0A0D0A2E6E61766261722D7269676874207B0D0A20202020666C6F61743A20726967687421696D706F7274616E743B0D0A7D0D0A0D0A2E6E61766261722D637573746F6D202E6E61766261722D6272616E6420696D67207B0D0A202020206D61782D77696474683A20313030253B0D0A202020206D61782D6865696768743A20313030253B0D0A7D0D0A;
      TEMP_6 : Array[1..1146] of Byte := 2F2A2043535320446F63756D656E74202A2F0D0A0D0A2E636F6C666F726D207B20666C6F61743A6C6566743B2077696474683A3530253B7D0D0A0D0A3A726F6F74207B0D0A202020202D2D636F6C6F722D677265656E3A20233030613837383B0D0A202020202D2D636F6C6F722D7265643A20236665356534313B0D0A202020202D2D636F6C6F722D627574746F6E3A20236664666666663B0D0A202020202D2D636F6C6F722D626C61636B3A20233030303B0D0A7D0D0A2E7377697463682D627574746F6E207B0D0A20202020646973706C61793A20696E6C696E652D626C6F636B3B0D0A7D0D0A2E7377697463682D627574746F6E202E7377697463682D627574746F6E5F5F636865636B626F78207B0D0A20202020646973706C61793A206E6F6E653B0D0A7D0D0A2E7377697463682D627574746F6E202E7377697463682D627574746F6E5F5F6C6162656C207B0D0A202020206261636B67726F756E642D636F6C6F723A20766172282D2D636F6C6F722D726564293B0D0A2020202077696474683A203472656D3B0D0A202020206865696768743A203272656D3B0D0A20202020626F726465722D7261646975733A203272656D3B0D0A20202020646973706C61793A20696E6C696E652D626C6F636B3B0D0A20202020706F736974696F6E3A2072656C61746976653B0D0A7D0D0A2E7377697463682D627574746F6E202E7377697463682D627574746F6E5F5F6C6162656C3A6265666F7265207B0D0A202020207472616E736974696F6E3A202E32733B0D0A20202020646973706C61793A20626C6F636B3B0D0A20202020706F736974696F6E3A206162736F6C7574653B0D0A2020202077696474683A203272656D3B0D0A202020206865696768743A203272656D3B0D0A202020206261636B67726F756E642D636F6C6F723A20766172282D2D636F6C6F722D627574746F6E293B0D0A20202020636F6E74656E743A2027273B0D0A20202020626F726465722D7261646975733A203530253B0D0A20202020626F782D736861646F773A20696E7365742030707820307078203070782031707820766172282D2D636F6C6F722D626C61636B293B0D0A7D0D0A2E7377697463682D627574746F6E202E7377697463682D627574746F6E5F5F636865636B626F783A636865636B6564202B202E7377697463682D627574746F6E5F5F6C6162656C207B0D0A202020206261636B67726F756E642D636F6C6F723A20766172282D2D636F6C6F722D677265656E293B0D0A7D0D0A2E7377697463682D627574746F6E202E7377697463682D627574746F6E5F5F636865636B626F783A636865636B6564202B202E7377697463682D627574746F6E5F5F6C6162656C3A6265666F7265207B0D0A202020207472616E73666F726D3A207472616E736C61746558283272656D293B0D0A7D0D0A2E636F6E7461696E65724872207B0D0A20202020646973706C61793A20666C65783B200D0A7D0D0A2E766572746963616C2D616C69676E207B0D0A20202020646973706C61793A20666C65783B0D0A20202020616C69676E2D6974656D733A2063656E7465723B0D0A7D;
   END_VAR
BEGIN
END_DATA_BLOCK

DATA_BLOCK "DB 335"   // DB335
{ S7_Optimized_Access := 'FALSE' }
AUTHOR : AWP_S7P
FAMILY : WEB
VERSION : 0.1
   VAR
      MAGIC : DWord := DW#16#4157_5046;
      CONSISTENCY_TAG : DWord := 616098220;
